{attribute addProperty BoxType "EL3423-0000-0020"}
{attribute addProperty Id "Active_EnergyAT %I*LINT648"}
{attribute addProperty CRC "551920714"}
{attribute addProperty SizeInBites "64"}
{attribute addProperty SizeInBytes "8"}
TYPE Total_Active_Reduced_20E5A44A :
STRUCT
	{attribute addProperty Name "Active_Energy"}
	Active_Energy AT %I* : LINT;
END_STRUCT
END_TYPE

(* stored: Version 1.2.0.0, ProductVersion 3.1.4024.9
   DUT Total_Active_Reduced_20E5A44A: Id {4e8cf3b7-748f-4ea2-878d-067374632d4d} *)
